SUBAPPLICATION Button_Method_IE (* VT-Button (Button_IE) ODER lokale argumentlose OPC-UA-Methode (ACTION=CREATE_METHOD, SERVER_0 - z.B. von Web-Client/Dashboard oder per CLIENT_0 von einer anderen Station aufgerufen) aktiviert -> 1 gemeinsames IND-Event. Analog zu Softkey_Aux_Method_IE, aber fuer einen regulaeren VT-Button statt SoftKey/AUX - herausgeloest aus logiBUS_AI_Calibrate_IDA_OPC (CO/CS kamen dort 2x identisch vor). *)
  (* Standard: 61499-2; Description: Copyright (c) 2026 Meisterschulen am Ostbahnhof This program and the accompanying materials are made available under the terms of the Eclipse Public License 2.0 which is available at https://www.eclipse.org/legal/epl-2.0/ SPDX-License-Identifier: EPL-2.0 *)
  (* Version 1.0, 2026-09-18, Franz Höpfinger, Meisterschulen am Ostbahnhof, initial implementation - herausgeloest aus logiBUS_AI_Calibrate_IDA_OPC (Button_IE + SERVER_0 + E_MERGE_2 kam dort 2x vor, fuer CO und CS), wiederverwendbar fuer jeden Event-Trigger, der per VT-Taste UND gleichberechtigt per Methode ausgeloest werden soll. *)
  PACKAGE MyLib::sys;
  IMPORT isobus::UT::io::Button::ButtonActivationCode::BT_PRESSED_LATCHED;
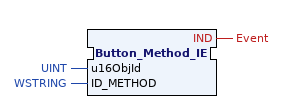
  EVENT_OUTPUT
    IND; (* Feuert wenn der Button ODER die lokale Methode aktiviert/aufgerufen wird *)
  END_EVENT
  VAR_INPUT
    u16ObjId : UINT; (* Object ID Button *)
    ID_METHOD : WSTRING; (* Lokale Methodenadresse (ACTION=CREATE_METHOD) fuer den argumentlosen Trigger - wird von Web-Client/Dashboard UND per CLIENT_0 von einer anderen Station aufgerufen *)
  END_VAR
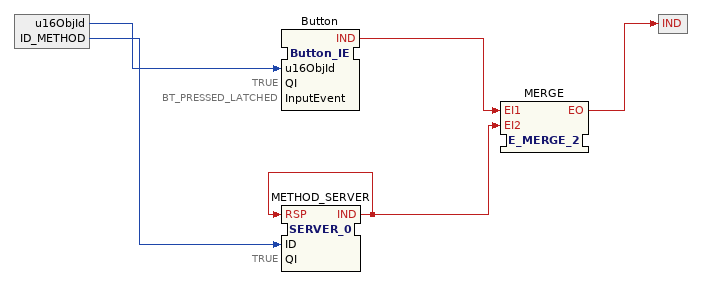
  (* RSP MUSS auf IND zurueckverdrahtet werden (argumentloser Trigger, keine Verarbeitung noetig) - sonst blockiert FORTEs onServerMethodCall den OPC-UA-Server-Thread bis zu 4s und haelt dabei open62541s globalen serviceMutex, den JEDER AX_PUBLISH_1 auf einem anderen FORTE-Thread ebenfalls braucht. Siehe Ventilsteuerung/OPC_UA_VERNETZUNG.md Punkt 12. *)
  FBS
    Button : isobus::UT::io::Button::Button_IE(QI := TRUE, InputEvent := BT_PRESSED_LATCHED);
    METHOD_SERVER : iec61499::net::SERVER_0(QI := TRUE);
    MERGE : iec61499::events::E_MERGE_2;
  END_FBS
  EVENT_CONNECTIONS
    Button.IND TO MERGE.EI1;
    METHOD_SERVER.IND TO MERGE.EI2;
    METHOD_SERVER.IND TO METHOD_SERVER.RSP;
    MERGE.EO TO IND;
  END_CONNECTIONS
  DATA_CONNECTIONS
    u16ObjId TO Button.u16ObjId;
    ID_METHOD TO METHOD_SERVER.ID;
  END_CONNECTIONS
END_SUBAPPLICATION
